# B&R Automation Studio project plcProject
Automation Studio 4.12.6.106

## Configuration Simulator

### Task classes (Cpu.sw)
```
Cyclic#1 (cycle 10000 us, tolerance 0 us):
  Logic <- Logic.prg
Binaries: vcnet, udbdef, vcrt, vcfntttf, FWRules, Hmi03, arial, vcmgr, vcpkat, vccovl, vccnum, vcpfar00, vcdsint, vcpdvnc, vcshared, vcpdsw, vcfile, vcalarm, vccbtn, vcgclass, vcdsloc, arialbd, Hmi02, Hmi01, TCData, vctcal, vccbmp, vcbclass, iomap, asfw, Role, sysconf, arconfig, ashwd, User, ashwac
Libraries: sys_lib, runtime, fileio, asieccon, dataobj, vcresman, astime, standard
```

### Hardware
```
PC : PC_any v1.1.1.0 (OrderNumber=PC)
  Connector IF3:
    Vnc1
    VncKeyMappingFile1 = VC\PS2-Keyboard.dis
    VncAuthentication1 = 1
    VncPasswordViewOnly1 = 0
    VncPasswordViewControl1 = 1
    VncRefreshRate1 = 100
  ConfigurationID = plcProject_Simulator
  SystemTick = 2000
  Cyclic1Duration = 10000
  Cyclic1Tolerance = 0
  FileDevice1
  FileDeviceName1 = USER
  FileDevicePath1 = USER_PATH
  ActivateOpcUa = 1
  OpcUaInformationModels_PV_Version = 1
```

## Logical view

### Program Logical/Logic

#### Types.typ
```iecst
TYPE
	Conveyor_Io_typ : 	STRUCT
		diPhotoeye1 : BOOL;
		diPhotoeye2 : BOOL;
		aoSpeed : REAL;
	END_STRUCT;
	Conveyor_Out_typ : 	STRUCT
		readyToSend : BOOL;
		readyToReceive : BOOL;
		transferComplete : BOOL;
	END_STRUCT;
	Conveyor_In_typ : 	STRUCT
		upstreamReadyToSend : BOOL;
		downstreamReadyToReceive : BOOL;
		beltSpeed : REAL;
	END_STRUCT;
	Conveyor_Internal_typ : 	STRUCT
		state : CONVEYOR_ST_enum;
	END_STRUCT;
	CONVEYOR_ST_enum :
		(
		CONVEYOR_ST_INIT,
		CONVEYOR_ST_READY_TO_RECEIVE,
		CONVEYOR_ST_RECEIVING,
		CONVEYOR_ST_POSITION,
		CONVEYOR_ST_READY_TO_SEND,
		CONVEYOR_ST_SENDING
		);
	Conveyor_typ : 	STRUCT
		in : Conveyor_In_typ;
		out : Conveyor_Out_typ;
		io : Conveyor_Io_typ;
		internal : Conveyor_Internal_typ;
	END_STRUCT;
END_TYPE
```

#### Variables.var
```iecst
VAR
	conveyor : ARRAY[0..MAI_CONVEYORS] OF Conveyor_typ;
END_VAR
VAR CONSTANT
	MAI_CONVEYORS : USINT := 4;
END_VAR
VAR
	index : USINT;
	processActive : BOOL;
END_VAR
```

#### Main.st
```iecst
PROGRAM _INIT

	FOR index := 0 TO MAI_CONVEYORS DO
		conveyor[index].in.beltSpeed := 1.4;
	END_FOR

	processTimer.PT := T#1.7s;

END_PROGRAM

PROGRAM _CYCLIC

	// Map conveyor outputs to neighboring conveyor inputs.
	conveyor[0].in.downstreamReadyToReceive := conveyor[1].out.readyToReceive;
	conveyor[0].in.upstreamReadyToSend := TRUE;
	conveyor[1].in.downstreamReadyToReceive := conveyor[2].out.readyToReceive;
	conveyor[1].in.upstreamReadyToSend := conveyor[0].out.readyToSend;
	conveyor[2].in.downstreamReadyToReceive := conveyor[3].out.readyToReceive;
	conveyor[2].in.upstreamReadyToSend := conveyor[1].out.readyToSend;
	conveyor[3].in.downstreamReadyToReceive := conveyor[4].out.readyToReceive;
	conveyor[3].in.upstreamReadyToSend := conveyor[2].out.readyToSend;
	conveyor[4].in.downstreamReadyToReceive := processTimer.Q;
	conveyor[4].in.upstreamReadyToSend := conveyor[3].out.readyToSend;

	FOR index := 0 TO MAI_CONVEYORS DO

		// Reset all output signal cyclically.
		conveyor[index].out.readyToReceive := FALSE;
		conveyor[index].out.readyToSend := FALSE;
		conveyor[index].out.transferComplete := FALSE;
		conveyor[index].io.aoSpeed := 0;

		CASE conveyor[index].internal.state OF

			CONVEYOR_ST_INIT:
				IF (conveyor[index].io.diPhotoeye2) THEN
					conveyor[index].internal.state := CONVEYOR_ST_READY_TO_SEND;
				ELSE
					conveyor[index].internal.state := CONVEYOR_ST_READY_TO_RECEIVE;
				END_IF

			CONVEYOR_ST_READY_TO_RECEIVE:
				conveyor[index].out.readyToReceive := TRUE;
				IF (conveyor[index].io.diPhotoeye1) THEN
					conveyor[index].internal.state := CONVEYOR_ST_RECEIVING;
				END_IF

			CONVEYOR_ST_RECEIVING:
				conveyor[index].out.readyToReceive := TRUE;
				conveyor[index].io.aoSpeed := conveyor[index].in.beltSpeed;
				IF (NOT conveyor[index].io.diPhotoeye1) THEN
					conveyor[index].internal.state := CONVEYOR_ST_POSITION;
				END_IF

			CONVEYOR_ST_POSITION:
				conveyor[index].io.aoSpeed := conveyor[index].in.beltSpeed;
				IF (conveyor[index].io.diPhotoeye2) THEN
					IF (conveyor[index].in.downstreamReadyToReceive) THEN
						conveyor[index].internal.state := CONVEYOR_ST_SENDING;
					ELSE
						conveyor[index].internal.state := CONVEYOR_ST_READY_TO_SEND;
					END_IF
				END_IF

			CONVEYOR_ST_READY_TO_SEND:
				conveyor[index].out.readyToSend := TRUE;
				IF (conveyor[index].in.downstreamReadyToReceive) THEN
					conveyor[index].internal.state := CONVEYOR_ST_SENDING;
				END_IF

			CONVEYOR_ST_SENDING:
				conveyor[index].out.readyToSend := TRUE;
				conveyor[index].io.aoSpeed := conveyor[index].in.beltSpeed;
				IF (NOT conveyor[index].io.diPhotoeye2) THEN
					conveyor[index].internal.state := CONVEYOR_ST_READY_TO_RECEIVE;
				END_IF

		END_CASE

	END_FOR

	// Handle process logic.
	processTimer.IN := conveyor[4].out.readyToSend;
	processTimer();
	processActive := processTimer.IN;

END_PROGRAM
```
